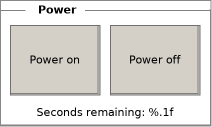
VISUALIZATION VISU_M2Power  // 212x127
VAR_IN_OUT
	ref : M2;
    widget : M2Widget;
END_VAR
    Polyline (85,10) (210,10) (210,125) (0,125) (0,10) (25,10)
    Label (35,0 45x20), "Power"
    Button (10,25 90x70), "Power on", input disabled if: ref.processes.powerOn.statuses.enabledStatus.disabled
        OnMouseClick: execute { ref.processes.powerOn.do_request := TRUE; }
    Button (110,25 90x70), "Power off", input disabled if: ref.processes.powerOff.statuses.enabledStatus.disabled
        OnMouseClick: execute { ref.processes.powerOff.do_request := TRUE; }
    Rectangle (10,100 190x25), "Seconds remaining: %.1f", text variable: ref.powerOffTimer
END_VISUALIZATION

(* stored: Version 1.1.0.1, ProductVersion 3.1.4018.5
   Visu VISU_M2Power: Id {5db2c0ab-b9a1-4958-9ffd-b73eb8706a60} *)
